% RSLogix 500 project I2P-JOB14-ADAM BOCZKIEWICZ_BAK061.RSS, saved by version 10.00.00.00 %
PROJECT "ML04A"    % processor: Bul.1763 MicroLogix 1100 Series B %

PROGRAM FILES
  LAD 2   14 rungs

DATA FILES
  O0 OUTPUT  4 elements
  I1 INPUT  6 elements
  S2 STATUS  66 elements
  B3 BINARY  1 elements
  T4 TIMER  1 elements
  C5 COUNTER  1 elements
  R6 CONTROL  1 elements
  N7 INTEGER  1 elements
  F8 FLOAT  1 elements

LADDER 2
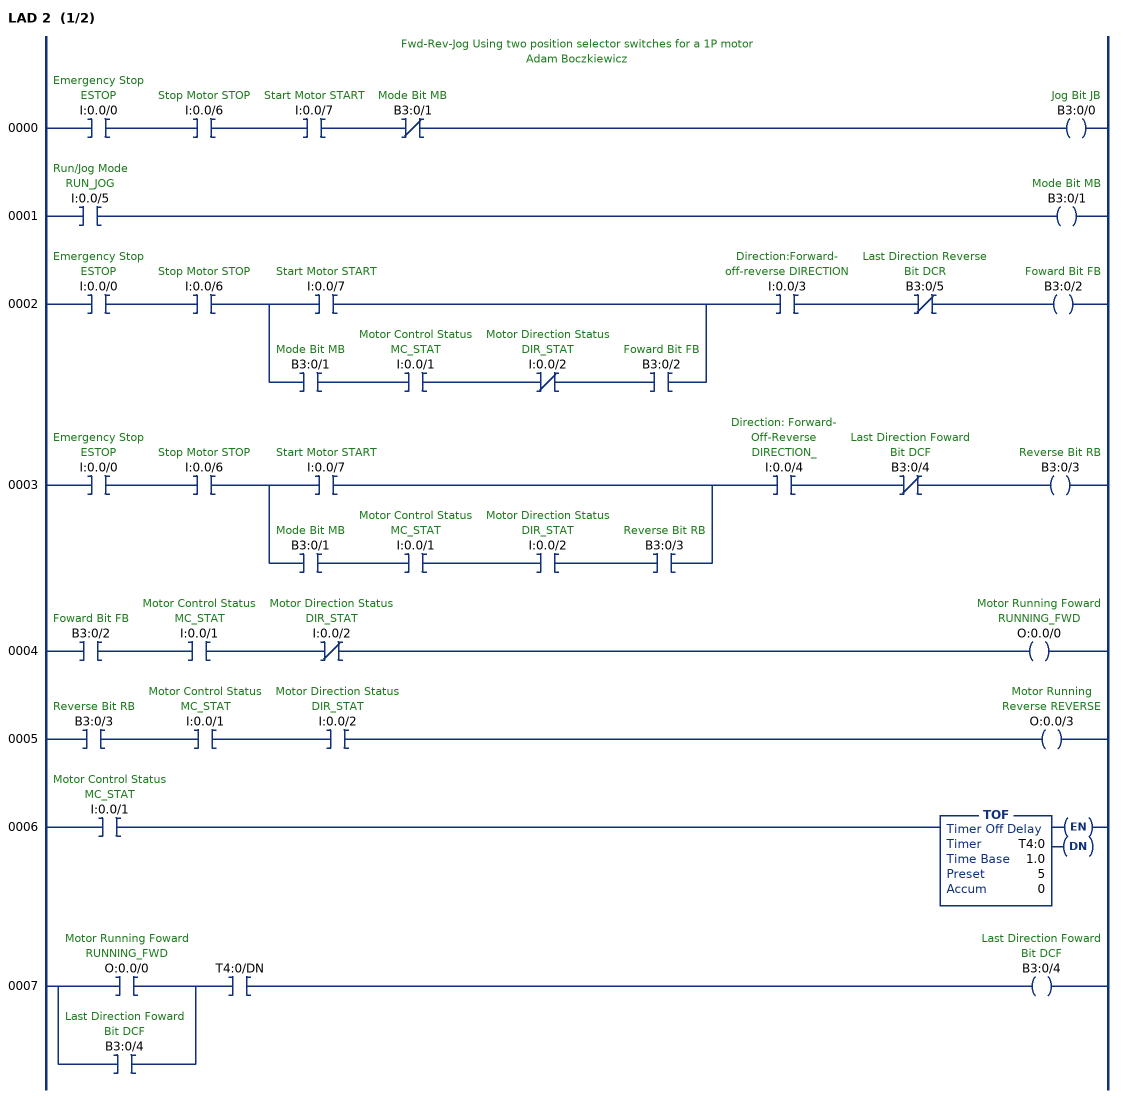
% Rung: 0 %
% Fwd-Rev-Jog Using two position selector switches for a 1P motor
% Adam Boczkiewicz %
SOR XIC I:0.0/0 XIC I:0.0/6 XIC I:0.0/7 XIO B3:0/1 OTE B3:0/0 EOR
%   I:0.0/0  ESTOP  "Emergency Stop" %
%   I:0.0/6  STOP  "Stop Motor" %
%   I:0.0/7  START  "Start Motor" %
%   B3:0/1  MB  "Mode Bit" %
%   B3:0/0  JB  "Jog Bit" %
% Rung: 1 %
SOR XIC I:0.0/5 OTE B3:0/1 EOR
%   I:0.0/5  RUN_JOG  "Run/Jog Mode" %
%   B3:0/1  MB  "Mode Bit" %
% Rung: 2 %
SOR XIC I:0.0/0 XIC I:0.0/6 BST XIC I:0.0/7 NXB XIC B3:0/1 XIC I:0.0/1 XIO I:0.0/2 XIC B3:0/2 BND XIC I:0.0/3 XIO B3:0/5 OTE B3:0/2 EOR
%   I:0.0/0  ESTOP  "Emergency Stop" %
%   I:0.0/6  STOP  "Stop Motor" %
%   I:0.0/7  START  "Start Motor" %
%   B3:0/1  MB  "Mode Bit" %
%   I:0.0/1  MC_STAT  "Motor Control Status" %
%   I:0.0/2  DIR_STAT  "Motor Direction Status" %
%   B3:0/2  FB  "Foward Bit" %
%   I:0.0/3  DIRECTION  "Direction:Forward- off-reverse" %
%   B3:0/5  DCR  "Last Direction Reverse Bit" %
% Rung: 3 %
SOR XIC I:0.0/0 XIC I:0.0/6 BST XIC I:0.0/7 NXB XIC B3:0/1 XIC I:0.0/1 XIC I:0.0/2 XIC B3:0/3 BND XIC I:0.0/4 XIO B3:0/4 OTE B3:0/3 EOR
%   I:0.0/0  ESTOP  "Emergency Stop" %
%   I:0.0/6  STOP  "Stop Motor" %
%   I:0.0/7  START  "Start Motor" %
%   B3:0/1  MB  "Mode Bit" %
%   I:0.0/1  MC_STAT  "Motor Control Status" %
%   I:0.0/2  DIR_STAT  "Motor Direction Status" %
%   B3:0/3  RB  "Reverse Bit" %
%   I:0.0/4  DIRECTION_  "Direction: Forward- Off-Reverse" %
%   B3:0/4  DCF  "Last Direction Foward Bit" %
% Rung: 4 %
SOR XIC B3:0/2 XIC I:0.0/1 XIO I:0.0/2 OTE O:0.0/0 EOR
%   B3:0/2  FB  "Foward Bit" %
%   I:0.0/1  MC_STAT  "Motor Control Status" %
%   I:0.0/2  DIR_STAT  "Motor Direction Status" %
%   O:0.0/0  RUNNING_FWD  "Motor Running Foward" %
% Rung: 5 %
SOR XIC B3:0/3 XIC I:0.0/1 XIC I:0.0/2 OTE O:0.0/3 EOR
%   B3:0/3  RB  "Reverse Bit" %
%   I:0.0/1  MC_STAT  "Motor Control Status" %
%   I:0.0/2  DIR_STAT  "Motor Direction Status" %
%   O:0.0/3  REVERSE  "Motor Running Reverse" %
% Rung: 6 %
SOR XIC I:0.0/1 TOF T4:0 1.0 5 0 EOR
%   I:0.0/1  MC_STAT  "Motor Control Status" %
% Rung: 7 %
SOR BST XIC O:0.0/0 NXB XIC B3:0/4 BND XIC T4:0/DN OTE B3:0/4 EOR
%   O:0.0/0  RUNNING_FWD  "Motor Running Foward" %
%   B3:0/4  DCF  "Last Direction Foward Bit" %

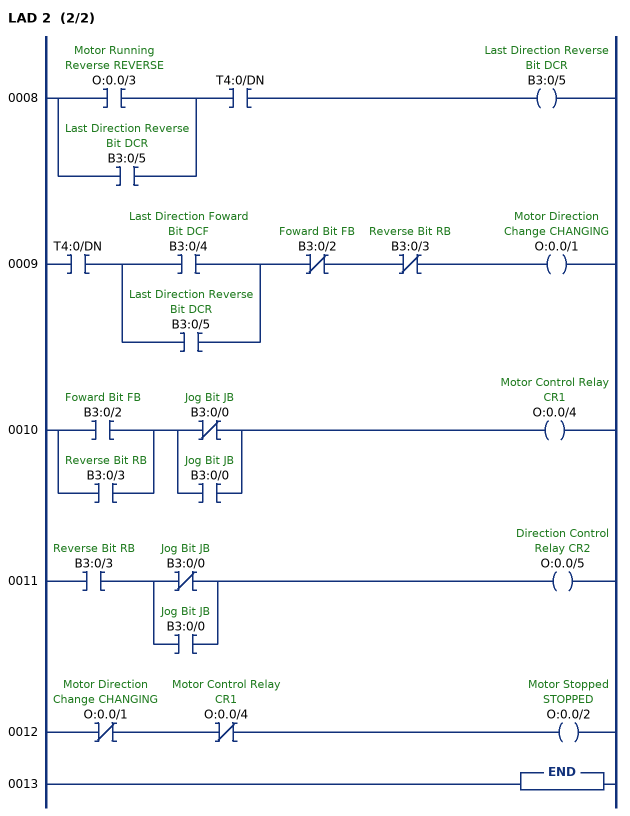
% Rung: 8 %
SOR BST XIC O:0.0/3 NXB XIC B3:0/5 BND XIC T4:0/DN OTE B3:0/5 EOR
%   O:0.0/3  REVERSE  "Motor Running Reverse" %
%   B3:0/5  DCR  "Last Direction Reverse Bit" %
% Rung: 9 %
SOR XIC T4:0/DN BST XIC B3:0/4 NXB XIC B3:0/5 BND XIO B3:0/2 XIO B3:0/3 OTE O:0.0/1 EOR
%   B3:0/4  DCF  "Last Direction Foward Bit" %
%   B3:0/5  DCR  "Last Direction Reverse Bit" %
%   B3:0/2  FB  "Foward Bit" %
%   B3:0/3  RB  "Reverse Bit" %
%   O:0.0/1  CHANGING  "Motor Direction Change" %
% Rung: 10 %
SOR BST XIC B3:0/2 NXB XIC B3:0/3 BND BST XIO B3:0/0 NXB XIC B3:0/0 BND OTE O:0.0/4 EOR
%   B3:0/2  FB  "Foward Bit" %
%   B3:0/3  RB  "Reverse Bit" %
%   B3:0/0  JB  "Jog Bit" %
%   O:0.0/4  CR1  "Motor Control Relay" %
% Rung: 11 %
SOR XIC B3:0/3 BST XIO B3:0/0 NXB XIC B3:0/0 BND OTE O:0.0/5 EOR
%   B3:0/3  RB  "Reverse Bit" %
%   B3:0/0  JB  "Jog Bit" %
%   O:0.0/5  CR2  "Direction Control Relay" %
% Rung: 12 %
SOR XIO O:0.0/1 XIO O:0.0/4 OTE O:0.0/2 EOR
%   O:0.0/1  CHANGING  "Motor Direction Change" %
%   O:0.0/4  CR1  "Motor Control Relay" %
%   O:0.0/2  STOPPED  "Motor Stopped" %
% Rung: 13 %
SOR END EOR

OTHER DOCUMENTED ADDRESSES
  I:0.0/8  REV  "Start Reverse"
  JOG  
  MO  
  T4:0/TT  TT

DATA TABLE (non-zero values as saved)
DATA T4
% .PRE .ACC %
% T4:0 % 5 0
DATA C5
% .PRE .ACC %
% C5:0 % 16 1
